PROGRAM MAIN
VAR
	bTest: BOOL;
	Ax1_FB_HomeBeforeMoveAX8000: FB_HomeBeforeMoveAX8000;
END_VAR
VAR PERSISTENT
	nTest : INT;
END_VAR

//Axis01
Axis01_Status();
Axis01_Interlock_ST();
Axis01_Command();
Axis01_Manual();
Axis01_Auto();
Axis01_Alarm();

//Axis02
Axis02_Status();
Axis02_Interlock_ST();
Axis02_Command();
Axis02_Manual();
Axis02_Auto();
Axis02_Alarm();
Axis02_Speed_Offset();
Axis02_Task_Offset();


//Axis03
Axis03_Status();
Axis03_Interlock_ST();
Axis03_Command();
Axis03_Manual();
Axis03_Auto();
Axis03_Alarm();

//Axis04
Axis04_Status();
Axis04_Command();
Axis04_Manual();
Axis04_Auto();
Axis04_Alarm();
Axis04_Set_Work_End_Speed();

//Axis05
Axis05_Interlock_ST();
Axis05_Alarm();
Axis05_Auto();
Axis05_Command();
Axis05_Manual();
Axis05_Status();

//Axis06
Axis06_Status();
Target_Distance();

//Alarm
Alarm_Error();
Alarm_Warring();

//System
HMI();
HOME_MOVE();
Initial();
Moving_Speed();
System();
Login_Timer();

//Vision
//Vision_ST();
Vision();
Move_Command();

//Work
Motion_Step_ST();
Vision_Step_ST();

END_PROGRAM

(* stored: Version 1.1.0.1, ProductVersion 3.1.4024.15
   POU MAIN: Id {6aabf998-5011-40c5-ad4e-540ab5ceb3b4}, SpecialFunc None *)
